{attribute 'linkalways'} 
{attribute 'no_explicit_call' := 'This FB is a CLASS and must be accessed using methods or properties'}
{attribute 'enable_dynamic_creation'}
FUNCTION_BLOCK Node_F_VN_CreateNDimensionalImage EXTENDS VisionNode
VAR
    ipImage : _ITcVnImage;
    aShape : _TcVnArray33_UDINT;
    ePixelType : _ETcVnElementType(ETcVnElementType.TCVN_ET_USINT);
    hrPrev : _HRESULT(S_OK);
	hresult : _HRESULT(S_OK);
END_VAR

METHOD PUBLIC  Clone : I_Node
VAR
	pNode : POINTER TO Node_F_VN_CreateNDimensionalImage;
END_VAR
pNode := __NEW(Node_F_VN_CreateNDimensionalImage);
Clone := pNode^;
END_METHOD

METHOD FB_init : BOOL
VAR_INPUT
	bInitRetains : BOOL; // if TRUE, the retain variables are initialized (warm start / cold start)
	bInCopyCode : BOOL;  // if TRUE, the instance afterwards gets moved into the copy code (online change)
END_VAR
AddParameter('aShape', aShape);
AddParameter('ePixelType', ePixelType);
AddInput('hrPrev', hrPrev);
AddOutput('ipImage', ipImage);
AddOutput('hresult',hresult);
END_METHOD

METHOD PROTECTED OnExecute
hresult.Value := F_VN_CreateNDimensionalImage(
    ipImage := ipImage.Value,
    aShape := aShape.Value,
    ePixelType := ePixelType.Value,
	hrPrev:= hrPrev.Value);
END_METHOD

METHOD PUBLIC PreExecutionCheck
VAR_INPUT
	Check : I_PreExecutionChecks;
END_VAR
END_METHOD

END_FUNCTION_BLOCK

(* stored: Version 1.1.0.1, ProductVersion 3.1.4024.13
   POU Node_F_VN_CreateNDimensionalImage: Id {eb23a248-f477-0b1f-0a41-25d5680551f6}, SpecialFunc None
   Folder Constructor: Id {b4778362-902f-0335-3d79-36b55252be3c}
   Method Clone: Id {643cea85-69a9-078e-3180-972074bdb7dd}
   Method FB_init: Id {60be2691-e9e9-03ec-00fe-989071b9260d}
   Method OnExecute: Id {a1659803-1b42-0f93-1f9b-f71a60711354}
   Method PreExecutionCheck: Id {fa038edb-e800-0909-3cb6-828631202b13} *)
